// TIA Portal V20 export
TYPE "LAxisCtrl_typePower"
TITLE = LAxisCtrl_typePower
// Support: tech.team.motioncontrol@siemens.com 
// Fax: +49 (0) 9131/98-1297
   STRUCT
      startMode : DInt := 1;   // 0: Enable axis not position-controlled; 1: Enable axis position-controlled (This parameter is ignored when a speed axis or external encoder is used)
      stopMode : Int := 0;   // 0: Emergency stop; 1: Immediate stop; 2: Stop with maximum dynamic values
      syncMotionSimulation : Bool := FALSE;   // TRUE: Start the simulation of synchronous operation automatically with falling edge at enableAxis; FALSE: No simulation of synchronous operation
   END_STRUCT;
END_TYPE
